// TIA Portal V15 export
// export: Created 2019-04-04T10:04:46.8154146Z, ExportSetting WithDefaults, WithReadOnly, DisplayName Totally Integrated Automation Portal, DisplayVersion V15, DisplayName TIA Portal Openness, DisplayVersion V15, DisplayName STEP 7 Professional, DisplayVersion V15, DisplayName STEP 7 Safety, DisplayVersion V15, DisplayName WinCC Professional, DisplayVersion V15, DisplayName SIMATIC Visualization Architect, DisplayVersion V15
FUNCTION "ROBNAME" : Void   // FC71, LAD
TITLE = Rob_ROBNAME
{ S7_Optimized_Access := 'TRUE' }
VERSION : 1.1
// stored: AutoNumber false, CodeModifiedDate 2019-04-04T10:04:01.8111922Z, CompileDate 2019-04-04T10:04:16.3409314Z, CreationDate 2019-04-04T10:03:42.2202115Z, HandleErrorsWithinBlock false, InterfaceModifiedDate 2017-06-20T14:56:00.5916118Z, IsConsistent true, IsIECCheckEnabled false, IsKnowHowProtected false, IsWriteProtected false, LibraryConformanceStatus The object is library-conformant., ModifiedDate 2019-04-04T10:04:01.8111922Z, ParameterModified 2017-06-20T14:56:00.5846118Z, PLCSimAdvancedSupport true, SetENOAutomatically False, StructureModified 2017-06-20T14:56:00.5916118Z, UDAEnableTagReadback false
   VAR_TEMP
      Temp : Struct
         _Bool : Bool;
         _Byte : Byte;
         _Word : Word;
         _DWord : DWord;
         _Int : Int;
         _DInt : DInt;
         _Real : Real;
         _S5Time : S5Time;
         _Time : Time;
      END_STRUCT;
   END_VAR
BEGIN
END_FUNCTION
